FUNCTION_BLOCK FB_NanotecPD_Move
VAR_INPUT
	bExecute 	: BOOL;
	bStop		: BOOL;
	nPosition	: DINT; //Reale Einheit (µm oder 1/10°)
	nSpeed		: DINT; //Reale Einheit/s	
END_VAR
VAR_OUTPUT
	bBusy 		: BOOL;
	bError 		: BOOL;
	nErrorId 	: ERRORID;	
END_VAR
VAR_IN_OUT
	pHwRef : POINTER TO FB_HwRefNanotecPD; 
END_VAR
VAR
	nState 					: USINT;
	eCurrentCoDS402State 	: E_CoDS402States;
	fbGetCurrTaskIndex		: GETCURTASKINDEX;
	nCurrentTaskCycleCount 	: UDINT;	
END_VAR

IF bExecute THEN
	eCurrentCoDS402State := pHwRef^.M_GetDS402State();
	
	CASE nState OF
		0:	//Vorbedingungen prüfen
			bBusy := TRUE;
			nState := 1;
			IF pHwRef^.bError THEN
				nErrorID := E_ErrorIdHwGeneral.ERRORID_DriveIsInErrorState;
				nState := 99;
			ELSE
				IF pHwRef^.bBusy THEN
					nErrorID := E_ErrorIdHwGeneral.ERRORID_DriveIsStillBusy;
					nState := 99;
				ELSE
					IF NOT pHwRef^.P_bIsHomed THEN
						nErrorID := E_ErrorIdHwGeneral.ERRORID_DriveNotHomed;
						nState := 99;
					ELSE
						IF NOT pHwRef^.M_SetTargetPos(nPosition) THEN
							nErrorID := E_ErrorIdHwGeneral.ERRORID_InvalidPosition;
							nState := 99;
						ELSE
							IF NOT pHwRef^.M_SetTargetSpeed(nSpeed) THEN
								nErrorID := E_ErrorIdHwGeneral.ERRORID_InvalidSpeed;
								nState := 99;
							END_IF
						END_IF	
					END_IF
				END_IF
			END_IF
			
			fbGetCurrTaskIndex();
			nCurrentTaskCycleCount := TwinCAT_SystemInfoVarList._TaskInfo[fbGetCurrTaskIndex.index].CycleCount;

		1:	//Mode sollte durch Homing bereits auf 1 stehen
			//Dieser State darf niemals im gleichen Zyklus wie State 0 ausgeführt werden. Passiert wenn FB im selben Zyklus auf-
			//gerufen wird. Somit wird sichergestellt, dass die Zielposition auch im Drive eher ankommt, wie das Startbit.
			IF TwinCAT_SystemInfoVarList._TaskInfo[fbGetCurrTaskIndex.index].CycleCount <> nCurrentTaskCycleCount THEN
				IF eCurrentCoDS402State = E_CoDS402States.DS402STATE_OperationEnabled THEN
					pHwRef^.nControlword := 31;
					nState := 2;
				ELSE
					nErrorID := E_ErrorIdDS402.ERRORID_OperationNotEnabled;
					nState := 99;
				END_IF
			END_IF
			
		2:	//Setpoint ACK?
			IF pHwRef^.nStatusword.12 THEN
				pHwRef^.nControlword := 15;
				nState := 3;
			END_IF
			
		3:	//Target reached?
			IF pHwRef^.bError THEN
				nErrorId := pHwRef^.P_nErrorID;
				nState := 99;
			ELSE
				{warning 'Safety sollte noch mit abgefragt werden'}
				IF bStop THEN
					pHwRef^.nControlword.8 := TRUE;
					nState := 4;
				END_IF
				
				IF pHwRef^.nStatusword.10 THEN
					nState := 80; //Ready
				END_IF
			END_IF
			
		4:	//Warten bis Motor sich nicht mehr dreht -> dann OperationEnable zurück nehmen
			IF pHwRef^.nCurrentSpeed = 0 THEN
				pHwRef^.nControlword := 7;
				nState := 5;
			END_IF			
			
		5:	//STM wieder in OperationEnable
			IF pHwRef^.M_GetDS402State() = E_CoDS402States.DS402STATE_SwitchedOn THEN
				pHwRef^.nControlword := 15;
				nState := 80; //Ready
			END_IF
	END_CASE
	
	IF nState >= 80 THEN
		bBusy := FALSE;
		IF nState = 99 THEN
			bError := TRUE;
		END_IF
	END_IF
	
ELSE
	bError := FALSE;
	nErrorId := 0;
	nState := 0;
END_IF

END_FUNCTION_BLOCK

(* stored: Version 1.1.0.1, ProductVersion 3.1.4024.11
   POU FB_NanotecPD_Move: Id {74970ab7-a201-4333-ad66-fd46e7033d18}, SpecialFunc None *)
